(* PLC project FromServer, Turbopneumatic Socket Server 1, author DVorobiev *)
(* stored: creationDateTime 2020-11-19T10:39:58, productRelease 1, companyURL www.turbo.ru, modificationDateTime 2020-12-23T15:55:29, version 1, organization Turbopneumatic *)

(* Create Call Socket class method *)
FUNCTION call_method : STRING
  VAR_INPUT
    id_Node : INT;
    nameFunction : STRING;
    id_Obj : INT;
    id_SubObj : INT;
    d_value : REAL;
  END_VAR

            call_method:=CONCAT(nameFunction,INT_TO_STRING(id_Node),',',INT_TO_STRING(id_Obj),',',REAL_TO_STRING(d_value),')');

          
END_FUNCTION

(* FB Socket.load_socket_node *)
FUNCTION_BLOCK load_socket_node
  VAR
    pyTrigger : BOOL;
    nameFunction : STRING := 'load_socket_node(';  (* Name Socket class method *)
  END_VAR
  VAR_INPUT
    id_Node : INT := 1;  (* Id for Node *)
    id_Obj : INT := 4096;  (* Id for Obj *)
    id_SubObj : INT := 0;  (* Id for SubObj *)
  END_VAR
  VAR
    python_eval0 : python_eval;
  END_VAR
  VAR_OUTPUT
    d_value : REAL;
  END_VAR
  VAR  (* added by the conversion: wires and edge detectors of the diagram *)
    _NOT2_OUT : BOOL;
  END_VAR

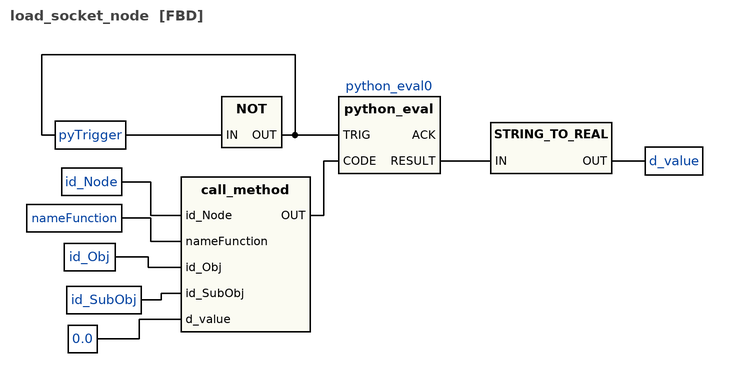
(* FBD diagram, written out as Structured Text *)
_NOT2_OUT := NOT pyTrigger;
pyTrigger := _NOT2_OUT;
python_eval0(TRIG := _NOT2_OUT, CODE := call_method(id_Node, nameFunction, id_Obj, id_SubObj, 0.0));
d_value := STRING_TO_REAL(python_eval0.RESULT);
END_FUNCTION_BLOCK

(* FB Socket.set_socket_node *)
FUNCTION_BLOCK set_socket_node
  VAR
    pyTrigger : BOOL;
    nameFunction : STRING := 'set_socket_node(';  (* Name Socket class method *)
  END_VAR
  VAR_INPUT
    id_Node : INT := 1;  (* Id for Node *)
    id_Obj : INT := 4097;  (* Id for Obj *)
    id_SubObj : INT := 0;  (* Id for SubObj *)
  END_VAR
  VAR
    python_eval0 : python_eval;
  END_VAR
  VAR_INPUT
    d_value : REAL;
  END_VAR
  VAR  (* added by the conversion: wires and edge detectors of the diagram *)
    _NOT2_OUT : BOOL;
  END_VAR

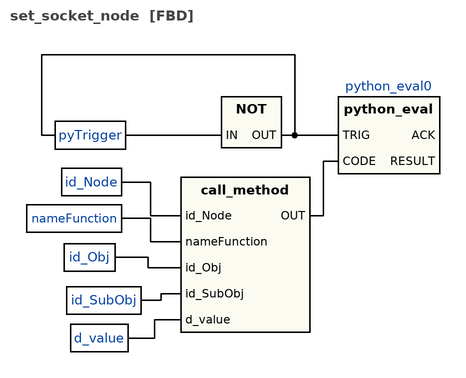
(* FBD diagram, written out as Structured Text *)
_NOT2_OUT := NOT pyTrigger;
pyTrigger := _NOT2_OUT;
python_eval0(TRIG := _NOT2_OUT, CODE := call_method(id_Node, nameFunction, id_Obj, id_SubObj, d_value));
END_FUNCTION_BLOCK

(* mainServer *)
PROGRAM test_1
  VAR
    id_Node : INT := 1;
    i_Obj : INT := 4096;
    i_Obj_1 : INT := 4097;
    i_SubObj : INT := 0;
    trigger0 : BOOL := False;
    s_out : STRING;
    d_value : REAL;
    d_val_out_1 : REAL;
    load_socket_node0 : load_socket_node;
    cycle : STRING := '0:0:1';
    set_socket_node0 : set_socket_node;
  END_VAR
  VAR  (* added by the conversion: wires and edge detectors of the diagram *)
    _EXPT31_OUT : ANY;
  END_VAR

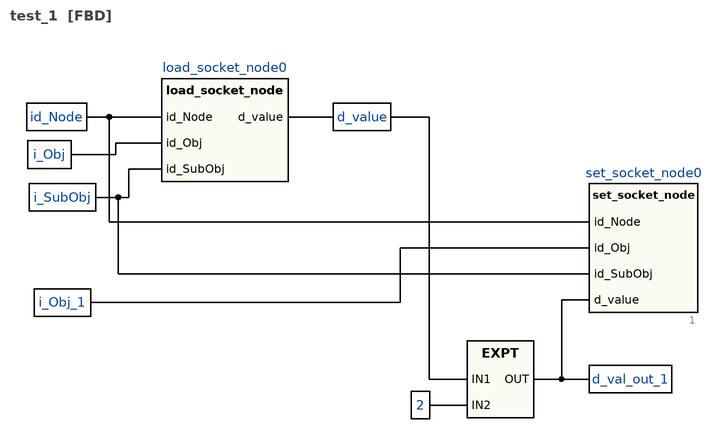
(* FBD diagram, written out as Structured Text *)
set_socket_node0(id_Node := id_Node, id_Obj := i_Obj_1, id_SubObj := i_SubObj, d_value := _EXPT31_OUT);
load_socket_node0(id_Node := id_Node, id_Obj := i_Obj, id_SubObj := i_SubObj);
d_value := load_socket_node0.d_value;
_EXPT31_OUT := EXPT(d_value, 2);
d_val_out_1 := _EXPT31_OUT;
END_PROGRAM

(* mainServer *)
PROGRAM mainServer
  VAR
    id_Node : INT := 1;
    i_Obj : INT := 4096;
    i_Obj_1 : INT := 4097;
    i_SubObj : INT := 0;
    trigger0 : BOOL := False;
    s_out : STRING;
    d_value : REAL;
    d_val_out_1 : REAL;
    load_socket_node0 : load_socket_node;
    INTEGRAL0 : INTEGRAL;
    cycle : STRING := '0:0:1';
    set_socket_node0 : set_socket_node;
  END_VAR
  VAR  (* added by the conversion: wires and edge detectors of the diagram *)
    _NOT14_OUT : BOOL;
  END_VAR

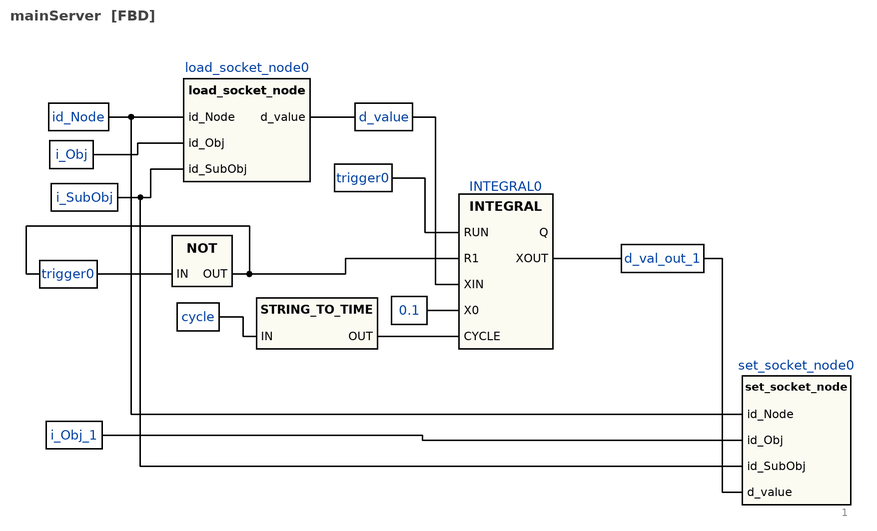
(* FBD diagram, written out as Structured Text *)
set_socket_node0(id_Node := id_Node, id_Obj := i_Obj_1, id_SubObj := i_SubObj, d_value := d_val_out_1);
load_socket_node0(id_Node := id_Node, id_Obj := i_Obj, id_SubObj := i_SubObj);
d_value := load_socket_node0.d_value;
_NOT14_OUT := NOT trigger0;
INTEGRAL0(RUN := trigger0, R1 := _NOT14_OUT, XIN := d_value, X0 := 0.1, CYCLE := STRING_TO_TIME(cycle));
d_val_out_1 := INTEGRAL0.XOUT;
trigger0 := _NOT14_OUT;
END_PROGRAM

CONFIGURATION config
  RESOURCE resource1 ON PLC
    TASK taskServer(INTERVAL := T#50ms, PRIORITY := 0);
    PROGRAM srv WITH taskServer : test_1;
  END_RESOURCE
END_CONFIGURATION
